PROGRAM MAIN
VAR
	Hearbeat				: DINT :=0;
	lrHotendTemp			: LREAL;
	bEnableExtrusionSystem 	: BOOL := FALSE;
	bResetExtrusionSystem 	: BOOL := FALSE;
	bEnableGimbalAxis 		: BOOL := TRUE;
	
	fUserOverride			: LREAL:= 100.0;
	in_stItpToPlc	AT %I*:	NcToPlc_NciChannel_Ref;
	out_stPlcToItp	AT %Q*:	PLCTONC_NCICHANNEL_REF;
	
	fbSimpleNciSequence		: FB_SimpleNciSequence;
	bExecSimpleNci:	BOOL	:= FALSE;
	
END_VAR

Hearbeat := Hearbeat+1;
GVL_IO.lrHotendTemp := GVL_IO.lrRawTemp/10.0;

PRG_ExtruderSys();

IF NOT  PRG_Init.BDONE THEN
	PRG_Init(bExecute:=TRUE , bDone=> );
	GVL_AxisCtrl.bEnableAxes := FALSE;

ELSE	(*Init done*)
		
	PRG_AxesEnable(
		//bEnable:= GVL_AxisCtrl.bEnableAxes,
		bEnable:= bEnableGimbalAxis,
		bHalt:= GVL_AxisCtrl.bHaltAxes,
		bReset:= GVL_AxisCtrl.bResetAxes,
		bAxesEnabled=> GVL_AxisCtrl.bRun, 
		bFaultActive=> , 
		wEnabledStates=> , 
		wFaultStates=> );
		
ItpSetOverridePercent(fOverridePercent:=fUserOverride , sPlcToNci:=out_stPlcToItp);

fbSimpleNciSequence(
	bExecute:= bExecSimpleNci, 
	bBusy=> , 
	bError=> , 
	bDone=> , 
	stX:=GVL_NC.Th1_AXIS, 
	stY:=GVL_NC.Th2_AXIS, 
	stZ:=GVL_NC.Th2_AXIS, 
	stItpToPlc:= in_stItpToPlc , 
	stPlcToItp:= out_stPlcToItp);		
END_IF;	
	
	
//PRG_ExtrusionSystem(
//	bEnable:= bEnableExtrusionSystem,
//	bReset := bResetExtrusionSystem);

END_PROGRAM

(* stored: Version 1.1.0.1, ProductVersion 3.1.4024.2
   POU MAIN: Id {0c1a4696-92e3-485c-8109-c9f8a167d8ed}, SpecialFunc None *)
